FUNCTION_BLOCK FB_ResetNC IMPLEMENTS I_Reset
VAR
    {attribute 'no_copy'}
    AxisRef : REFERENCE TO AXIS_REF;
    fbMcReset 	: MC_Reset;
END_VAR

IF NOT __ISVALIDREF(AxisRef) THEN
    RETURN;
END_IF

fbMcReset( Axis := AxisRef );

PROPERTY Aborted : BOOL
GET
END_GET
END_PROPERTY

PROPERTY Active : BOOL
GET
END_GET
END_PROPERTY

PROPERTY Busy : BOOL
GET
Busy := THIS^.fbMcReset.Busy;
END_GET
END_PROPERTY

METHOD PUBLIC CallAfterInit
VAR_INPUT
    AxisRef : REFERENCE TO AXIS_REF;
END_VAR
THIS^.AxisRef REF= AxisRef;
END_METHOD

PROPERTY Done : BOOL
GET
Done := THIS^.fbMcReset.Done;
END_GET
END_PROPERTY

PROPERTY Error : BOOL
GET
Error := THIS^.fbMcReset.Error;
END_GET
END_PROPERTY

PROPERTY ErrorID : UDINT
GET
ErrorID := THIS^.fbMcReset.ErrorID;
END_GET
END_PROPERTY

METHOD FB_Init : BOOL
VAR_INPUT
    bInitRetains : BOOL; // if TRUE, the retain variables are initialized (warm start / cold start)
    bInCopyCode : BOOL;  // if TRUE, the instance afterwards gets moved into the copy code (online change)
    AxisRef : REFERENCE TO AXIS_REF;
END_VAR
THIS^.AxisRef REF= AxisRef;
END_METHOD

PROPERTY Message : T_MAXSTRING
GET
END_GET
END_PROPERTY

METHOD Reset
VAR_INPUT
END_VAR
// Clear previous status
fbMcReset(Execute := FALSE,  Axis := THIS^.AxisRef);
// initiate a new Resetting request
fbMcReset(   Axis := THIS^.AxisRef,
             Execute := TRUE );
END_METHOD

METHOD ResetDone
// Clear previous status
fbMcReset(Execute := FALSE,  Axis := THIS^.AxisRef);
END_METHOD

END_FUNCTION_BLOCK

(* stored: Version 1.1.0.1
   POU FB_ResetNC: Id {d5a33439-9af6-4b4b-814e-6ef8d170f497}, SpecialFunc None
   Property Aborted: Id {2aa8b146-892b-4eda-90ec-32907f9020a6}
   Get Get: Id {236b2987-0f8e-4912-a72b-8f244392ed75}
   Property Active: Id {afb1cb16-ce6f-476a-872b-292391db0ba9}
   Get Get: Id {5ec9be53-31c3-46c8-9997-d5f8c475074f}
   Property Busy: Id {5f2cceba-7134-4efe-8841-ecba923dca52}
   Get Get: Id {85f46149-33a8-4c33-ba36-19cb1218e31e}
   Method CallAfterInit: Id {771e705c-7d5a-4ab1-a753-7d7642187d6b}
   Property Done: Id {83716cc5-e3e4-4a0e-9a01-85c819af47e4}
   Get Get: Id {d0f9a103-0936-46aa-8fa2-cde1fa260a72}
   Property Error: Id {78cdb70e-09fe-40ab-8a68-7cb4953ca907}
   Get Get: Id {2ba6de77-2d92-47f3-802e-65abb1e872ab}
   Property ErrorID: Id {bfe921c1-e744-48fe-ba23-596c2a44a3af}
   Get Get: Id {50a11289-cfb4-4cf4-a1ea-ea391b17d488}
   Method FB_Init: Id {0ffde760-6475-4a6a-8e1c-babbb252f4cc}
   Property Message: Id {a5706ef5-f74c-4bf4-9005-1b34aba004a5}
   Get Get: Id {e44fad7f-c952-4ca6-9097-837dc45b6378}
   Method Reset: Id {b05fc0aa-59e5-483e-8e1e-55eb45708bf0}
   Method ResetDone: Id {703d31eb-b69f-4e59-82a6-fb6d1d408441} *)
